{attribute 'GeneratedUsingTerminal: EL9222-4433-0018'}
{attribute addProperty BoxType "EL9222-4433-0018"}
{attribute addProperty Id "OCP_Inputs_Channel_1AT %I*OCP_Inputs_Channel_8CCE65FB11OCP_Inputs_Channel_2AT %I*OCP_Inputs_Channel_8CCE65FB11OCP_Outputs_Channel_1AT %Q*OCP_Outputs_Channel_010149342OCP_Outputs_Channel_2AT %Q*OCP_Outputs_Channel_010149342WcStateAT %I*WcState_9091E0EB2InfoDataAT %I*InfoData_94A18F5E2"}
{attribute addProperty CRC "3683641335"}
{attribute addProperty Size "30"}
TYPE EL9222_DB8FE7F7 EXTENDS EtcSlaveTerminalBase_947E5A46 :
STRUCT
	{attribute addProperty Name "OCP_Inputs_Channel_1"}
	OCP_Inputs_Channel_1 : OCP_Inputs_Channel_8CCE65FB;
	{attribute addProperty Name "OCP_Inputs_Channel_2"}
	OCP_Inputs_Channel_2 : OCP_Inputs_Channel_8CCE65FB;
	{attribute addProperty Name "OCP_Outputs_Channel_1"}
	OCP_Outputs_Channel_1 : OCP_Outputs_Channel_01014934;
	{attribute addProperty Name "OCP_Outputs_Channel_2"}
	OCP_Outputs_Channel_2 : OCP_Outputs_Channel_01014934;
	{attribute addProperty Name "WcState"}
	WcState : WcState_9091E0EB;
	{attribute addProperty Name "InfoData"}
	InfoData : InfoData_94A18F5E;
END_STRUCT
END_TYPE

(* stored: Version 1.2.0.0, ProductVersion 3.1.4024.9
   DUT EL9222_DB8FE7F7: Id {b92de167-3214-4cf8-b1ce-a5f871aef7ad} *)
